// TIA Portal project "Program_Integration_S7-1500xIV3" (V15.1)

(* hardware
DEVICE "S71500/ET200MP station_1"  S7-1500 station
   slot 0: "Rail_0"  Rack  6ES7 590-1***0-0AA0
   slot 1: "PLC_1"  CPU 1515F-2 PN  6ES7 515-2FM01-0AB0  V2.6
      slot 3: "CPU display_1"  6ES7591-1BA00-0AA0
DEVICE "IV3-600CA"  GSD.Device.PN
   slot 0: "Rack"  Rack  V1.0
   slot 0: "IV3-600CA"  IV3-XXXX  IV3-XXXX  V1.0.0
      slot 0: "IV3-XXXX"  IV3-XXXX  1.0
      slot 1: "Interface"  Interface
         slot 1: "Port 1"  Port 1
   slot 1: "Command Control_1"  Command Control
      slot 0: "Command Control"  Command Control
   slot 2: "Command Status Bits_1"  Command Status Bits
      slot 0: "Command Status Bits"  Command Status Bits
   slot 3: "Device Result Bits_1"  Device Result Bits
      slot 0: "Device Result Bits"  Device Result Bits
   slot 4: "Device Status Words_1"  Device Status Words
      slot 0: "Device Status Words"  Device Status Words
   slot 5: "Device Statistics_1"  Device Statistics
      slot 0: "Device Statistics"  Device Statistics
   slot 6: "Position Adjust Result_1"  Position Adjust Result
      slot 0: "Position Adjust Result"  Position Adjust Result
   slot 7: "Tool Result_1"  Tool Result
      slot 0: "Tool Result"  Tool Result
   slot 8: "Tool Result_2"  Tool Result
      slot 0: "Tool Result"  Tool Result
   slot 9: "Tool Result_3"  Tool Result
      slot 0: "Tool Result"  Tool Result
   slot 10: "Tool Result_4"  Tool Result
      slot 0: "Tool Result"  Tool Result
   slot 11: "Tool Result_5"  Tool Result
      slot 0: "Tool Result"  Tool Result
   slot 12: "Tool Result_6"  Tool Result
      slot 0: "Tool Result"  Tool Result
   slot 13: "Tool Result_7"  Tool Result
      slot 0: "Tool Result"  Tool Result
   slot 14: "Tool Result_8"  Tool Result
      slot 0: "Tool Result"  Tool Result
   slot 15: "Tool Result_9"  Tool Result
      slot 0: "Tool Result"  Tool Result
   slot 16: "Tool Result_10"  Tool Result
      slot 0: "Tool Result"  Tool Result
   slot 17: "Tool Result_11"  Tool Result
      slot 0: "Tool Result"  Tool Result
   slot 18: "Tool Result_12"  Tool Result
      slot 0: "Tool Result"  Tool Result
   slot 19: "Tool Result_13"  Tool Result
      slot 0: "Tool Result"  Tool Result
   slot 20: "Tool Result_14"  Tool Result
      slot 0: "Tool Result"  Tool Result
   slot 21: "Tool Result_15"  Tool Result
      slot 0: "Tool Result"  Tool Result
   slot 22: "Tool Result_16"  Tool Result
      slot 0: "Tool Result"  Tool Result
   slot 23: "Tool Result_17"  Tool Result
      slot 0: "Tool Result"  Tool Result
   slot 24: "Tool Result_18"  Tool Result
      slot 0: "Tool Result"  Tool Result
   slot 25: "Tool Result_19"  Tool Result
      slot 0: "Tool Result"  Tool Result
   slot 26: "Tool Result_20"  Tool Result
      slot 0: "Tool Result"  Tool Result
   slot 27: "Tool Result_21"  Tool Result
      slot 0: "Tool Result"  Tool Result
   slot 28: "Tool Result_22"  Tool Result
      slot 0: "Tool Result"  Tool Result
   slot 29: "Tool Result_23"  Tool Result
      slot 0: "Tool Result"  Tool Result
   slot 30: "Tool Result_24"  Tool Result
      slot 0: "Tool Result"  Tool Result
   slot 31: "Tool Result_25"  Tool Result
      slot 0: "Tool Result"  Tool Result
   slot 32: "Tool Result_26"  Tool Result
      slot 0: "Tool Result"  Tool Result
   slot 33: "Tool Result_27"  Tool Result
      slot 0: "Tool Result"  Tool Result
   slot 34: "Tool Result_28"  Tool Result
      slot 0: "Tool Result"  Tool Result
   slot 35: "Tool Result_29"  Tool Result
      slot 0: "Tool Result"  Tool Result
   slot 36: "Tool Result_30"  Tool Result
      slot 0: "Tool Result"  Tool Result
   slot 37: "Tool Result_31"  Tool Result
      slot 0: "Tool Result"  Tool Result
   slot 38: "Tool Result_32"  Tool Result
      slot 0: "Tool Result"  Tool Result
   slot 39: "Tool Result_33"  Tool Result
      slot 0: "Tool Result"  Tool Result
   slot 40: "Tool Result_34"  Tool Result
      slot 0: "Tool Result"  Tool Result
   slot 41: "Tool Result_35"  Tool Result
      slot 0: "Tool Result"  Tool Result
   slot 42: "Tool Result_36"  Tool Result
      slot 0: "Tool Result"  Tool Result
   slot 43: "Tool Result_37"  Tool Result
      slot 0: "Tool Result"  Tool Result
   slot 44: "Tool Result_38"  Tool Result
      slot 0: "Tool Result"  Tool Result
   slot 45: "Tool Result_39"  Tool Result
      slot 0: "Tool Result"  Tool Result
   slot 46: "Tool Result_40"  Tool Result
      slot 0: "Tool Result"  Tool Result
   slot 47: "Tool Result_41"  Tool Result
      slot 0: "Tool Result"  Tool Result
   slot 48: "Tool Result_42"  Tool Result
      slot 0: "Tool Result"  Tool Result
   slot 49: "Tool Result_43"  Tool Result
      slot 0: "Tool Result"  Tool Result
   slot 50: "Tool Result_44"  Tool Result
      slot 0: "Tool Result"  Tool Result
   slot 51: "Tool Result_45"  Tool Result
      slot 0: "Tool Result"  Tool Result
   slot 52: "Tool Result_46"  Tool Result
      slot 0: "Tool Result"  Tool Result
   slot 53: "Tool Result_47"  Tool Result
      slot 0: "Tool Result"  Tool Result
   slot 54: "Tool Result_48"  Tool Result
      slot 0: "Tool Result"  Tool Result
   slot 55: "Tool Result_49"  Tool Result
      slot 0: "Tool Result"  Tool Result
   slot 56: "Tool Result_50"  Tool Result
      slot 0: "Tool Result"  Tool Result
   slot 57: "Tool Result_51"  Tool Result
      slot 0: "Tool Result"  Tool Result
   slot 58: "Tool Result_52"  Tool Result
      slot 0: "Tool Result"  Tool Result
   slot 59: "Tool Result_53"  Tool Result
      slot 0: "Tool Result"  Tool Result
   slot 60: "Tool Result_54"  Tool Result
      slot 0: "Tool Result"  Tool Result
   slot 61: "Tool Result_55"  Tool Result
      slot 0: "Tool Result"  Tool Result
   slot 62: "Tool Result_56"  Tool Result
      slot 0: "Tool Result"  Tool Result
   slot 63: "Tool Result_57"  Tool Result
      slot 0: "Tool Result"  Tool Result
   slot 64: "Tool Result_58"  Tool Result
      slot 0: "Tool Result"  Tool Result
   slot 65: "Tool Result_59"  Tool Result
      slot 0: "Tool Result"  Tool Result
   slot 66: "Tool Result_60"  Tool Result
      slot 0: "Tool Result"  Tool Result
   slot 67: "Tool Result_61"  Tool Result
      slot 0: "Tool Result"  Tool Result
   slot 68: "Tool Result_62"  Tool Result
      slot 0: "Tool Result"  Tool Result
   slot 69: "Tool Result_63"  Tool Result
      slot 0: "Tool Result"  Tool Result
   slot 70: "Tool Result_64"  Tool Result
      slot 0: "Tool Result"  Tool Result
   slot 71: "Device Result Bits_2"  Device Result Bits
      slot 0: "Device Result Bits"  Device Result Bits
*)

// ===== PLC "PLC_1"  CPU 1515F-2 PN =====
// protected blocks, not shown: "Main_Safety_RTG1", "Main_Safety_RTG1_DB"

VAR_GLOBAL   // PLC tag table "IV3 Tag"
   "Trigger request" AT %Q0.0 : Bool;
   "Programm switching request" AT %Q0.2 : Bool;
   "RUN" AT %I2.4 : Bool;
   "Ready" AT %I2.5 : Bool;
   "Busy" AT %I2.2 : Bool;
   "Overall judgement NG" AT %I4.6 : Bool;
   "Overall judgment OK" AT %I4.0 : Bool;
   "Logic 1" AT %I4.2 : Bool;
   "Logic 2" AT %I4.3 : Bool;
   "Logic 3" AT %I4.4 : Bool;
   "Logic 4" AT %I4.5 : Bool;
   "Trigger response" AT %I0.0 : Bool;
   "Memory status NG" AT %M20.1 : Bool;
   "Programm No." AT %QW4 : Word;
   "program change response" AT %I0.2 : Bool;
   "Program atual" AT %QB5 : Byte;
   "Alarme HMI receita" AT %M20.3 : Bool;
   "Start" AT %M15.0 : Bool;
   "SwitchToNamber" AT %MW4 : Word;
   "Memory status OK" AT %M12.5 : Bool;
   "Start program 3" AT %M29.0 : Bool;
   "Trigger troca" AT %M29.1 : Bool;
   "START TRIGG" AT %M29.2 : Bool;
   "Busy Start" AT %M12.2 : Bool;
   "Program 1" AT %M30.0 : Bool;
   "Program 2" AT %M30.1 : Bool;
   "Program 3" AT %M30.2 : Bool;
   "Error" AT %I3.7 : Bool;
END_VAR

DATA_BLOCK "IV3 Program_DB_1"   // DB2
{ S7_Optimized_Access := 'TRUE' }
VERSION : 0.1
// stored: InstanceOfName IV3 Program
"IV3 Program"
BEGIN
END_DATA_BLOCK

FUNCTION_BLOCK "IV3 Program"   // FB5, LAD
{ S7_Optimized_Access := 'TRUE' }
VERSION : 0.1
// TRATA SOLICITACAO DE TROCA DO PROGRAMA DO IV3 COM A RECEITA SELECIONADA NA HMI
   VAR_IN_OUT
      "Mov Req" : Bool;
      "Switch Req" : Bool;
   END_VAR
   VAR_TEMP   // added for the SCL form of the ladder/FBD networks
      _w1 : Bool;
   END_VAR
BEGIN

REGION Network 1: START MEMORY PULSO PROGRAM
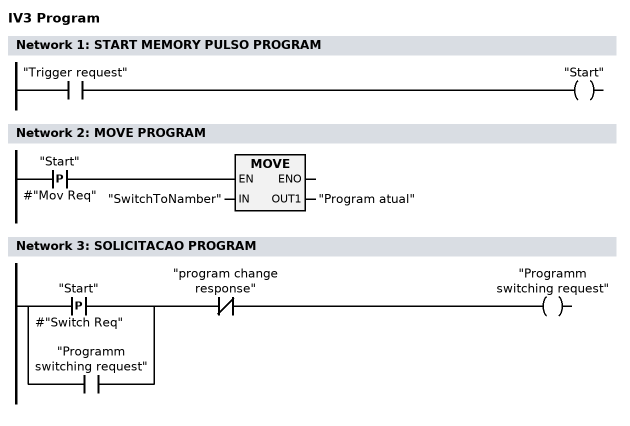
   RUNG wire#powerrail
      Contact( "Trigger request" )
      Coil( "Start" )
   END_RUNG
   // the same network as SCL:
   "Start" := "Trigger request";
END_REGION

REGION Network 2: MOVE PROGRAM
   RUNG wire#powerrail
      P_Contact(operand := "Start", bit := #"Mov Req")
      Move(in := "SwitchToNamber", out1 => "Program atual")
   END_RUNG
   // the same network as SCL:
   #_w1 := "Start" AND NOT #"Mov Req";   // rising edge of "Start"
   #"Mov Req" := "Start";
   IF #_w1 THEN "Program atual" := "SwitchToNamber"; END_IF;
END_REGION

REGION Network 3: SOLICITACAO PROGRAM
   RUNG wire#powerrail
      P_Contact(operand := "Start", bit := #"Switch Req")
      wire#w1
      I_Contact( "program change response" )
      Coil( "Programm switching request" )
   END_RUNG
   RUNG wire#powerrail
      Contact( "Programm switching request" )
   END_RUNG wire#w1
   // the same network as SCL:
   #_w1 := "Start" AND NOT #"Switch Req";   // rising edge of "Start"
   #"Switch Req" := "Start";
   "Programm switching request" := (#_w1 OR "Programm switching request") AND NOT "program change response";
END_REGION
END_FUNCTION_BLOCK

FUNCTION "IV3" : Void   // FC13, LAD
TITLE = FC DEDICADA PARA O SENSOR DE VISAO IV3
{ S7_Optimized_Access := 'TRUE' }
VERSION : 0.1
BEGIN

REGION Network 1: REQUISICAO PARA DISPARO IV3
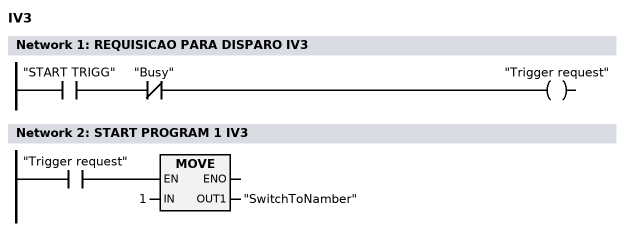
   RUNG wire#powerrail
      Contact( "START TRIGG" )
      I_Contact( "Busy" )
      Coil( "Trigger request" )
   END_RUNG
   // the same network as SCL:
   "Trigger request" := "START TRIGG" AND NOT "Busy";
END_REGION

REGION Network 2: START PROGRAM 1 IV3
   RUNG wire#powerrail
      Contact( "Trigger request" )
      Move(in := 1, out1 => "SwitchToNamber")
   END_RUNG
   // the same network as SCL:
   IF "Trigger request" THEN "SwitchToNamber" := 1; END_IF;
END_REGION
END_FUNCTION

ORGANIZATION_BLOCK "Main"   // OB1, LAD, ProgramCycle
TITLE = "Main Program Sweep (Cycle)"
{ S7_Optimized_Access := 'TRUE' }
VERSION : 0.1
   VAR_INPUT
      Initial_Call : Bool;   // Initial call of this OB
      Remanence : Bool;   // =True, if remanent data are available
   END_VAR
BEGIN

REGION Network 1: Chamada da FC13
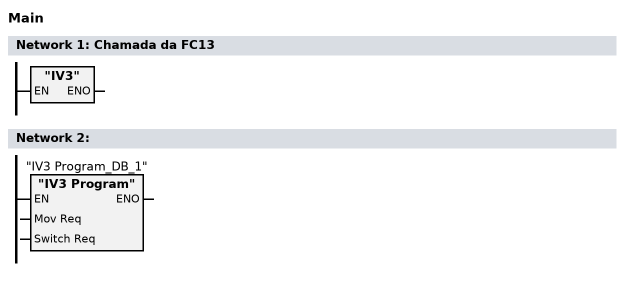
   RUNG wire#powerrail
      "IV3"()
   END_RUNG
   // the same network as SCL:
   "IV3"();
END_REGION

REGION Network 2
   RUNG wire#powerrail
      "IV3 Program_DB_1"("Mov Req" :=, "Switch Req" :=)
   END_RUNG
   // the same network as SCL:
   "IV3 Program_DB_1"();   // "IV3 Program"
END_REGION
END_ORGANIZATION_BLOCK